{attribute 'linkalways'} 
{attribute 'no_explicit_call' := 'This FB is a CLASS and must be accessed using methods or properties'}
{attribute 'enable_dynamic_creation'}
FUNCTION_BLOCK ChunkedRequest EXTENDS Disposable IMPLEMENTS I_Request
VAR
	request : I_Request;
	chunkedRequestData : REFERENCE TO I_ChunkedRequestSessionData;
END_VAR

PROPERTY PUBLIC CreatedTimestamp : I_Timestamp
GET
CreatedTimestamp := request.CreatedTimestamp;
END_GET
END_PROPERTY

METHOD FB_init : BOOL
VAR_INPUT
	bInitRetains : BOOL; // if TRUE, the retain variables are initialized (warm start / cold start)
	bInCopyCode : BOOL;  // if TRUE, the instance afterwards gets moved into the copy code (online change)
	Request : I_Request;
	ChunkedRequestData : Reference to I_ChunkedRequestSessionData;
END_VAR
THIS^.request := Request;
this^.chunkedRequestData ref= ChunkedRequestData;
END_METHOD

PROPERTY PUBLIC Header : I_Header
GET
Header := request.Header;
END_GET
END_PROPERTY

PROPERTY PUBLIC PayloadAddress : POINTER TO STRING
GET
IF chunkedRequestData = 0 THEN
	RETURN;
END_IF

PayloadAddress := chunkedRequestData.PayloadAddress;
END_GET
END_PROPERTY

PROPERTY PUBLIC PayloadSizeInBytes : UDINT
GET
IF chunkedRequestData = 0 THEN
	RETURN;
END_IF

PayloadSizeInBytes := chunkedRequestData.PayloadSizeInBytes;
END_GET
END_PROPERTY

END_FUNCTION_BLOCK

(* stored: Version 1.1.0.1, ProductVersion 3.1.4024.12
   POU ChunkedRequest: Id {aa683a94-86ec-4308-aa1b-d03a81190df9}, SpecialFunc None
   Folder Constructor: Id {34f599f7-f374-4a8a-9c64-52b4fd0e6efb}
   Property CreatedTimestamp: Id {744ce470-09e6-47ef-a611-4174f8540a99}
   Get Get: Id {11a617cf-3439-470f-b18b-9c8d1d2cfb11}
   Method FB_init: Id {08e94978-5994-40ad-8a88-96ed8acc840f}
   Property Header: Id {010e3e42-9687-478a-b993-1d469bcbbd40}
   Get Get: Id {c774c5c7-659e-42c1-afc5-0dda09dc5780}
   Property PayloadAddress: Id {590d487c-482d-4821-929f-d015aa0928c7}
   Get Get: Id {f0cfe211-405d-461e-88a4-a82378e44f5a}
   Property PayloadSizeInBytes: Id {833802e1-0b66-4074-8b68-674922585b9c}
   Get Get: Id {e889ed60-b02a-4a68-98c3-4df7aa0d693d} *)
